TYPE HMI_ERR_General :
STRUCT
	//General IO
	//prio's: emergency stop items == 100, e-circuit=99, default (nothing specified) = 50
	//adjust as needed
	ExampleErrorPreConfiggedPrio:BOOL;					//Error[prio=90] Example error with preconfigured prio (key only used at first creation/adding to the HMI-alarm-list-file)
END_STRUCT
END_TYPE

(* stored: Version 1.1.0.1
   DUT HMI_ERR_General: Id {a39dcdd6-6984-4217-9f7c-62f8eb1a63fa} *)
